// TIA Portal V16 export
// export: Created 2024-12-03T15:41:41.2290419Z, ExportSetting WithDefaults, DisplayName Totally Integrated Automation Portal, DisplayVersion V16 Update 6, DisplayName TIA Portal Version Control Interface, DisplayVersion V16 Update 2, DisplayName TIA Portal Openness, DisplayVersion V16 Update 6, DisplayName TIA Portal Teamcenter Gateway, DisplayVersion V16, DisplayName SINAMICS Startdrive Advanced, DisplayVersion V16 Update 5, DisplayName SINAMICS Startdrive G130, G150, S120, S150, SINAMICS MV, S210, DisplayVersion V16 Update 5, DisplayName SINAMICS Startdrive G110M, G120, G120C, G120D, G120P, G115D, DisplayVersion V16 Update 5, DisplayName STEP 7 Professional, DisplayVersion V16 Update 6, DisplayName STEP 7 Safety, DisplayVersion V16, DisplayName WinCC Advanced / Unified PC, DisplayVersion V16 Update 6
FUNCTION_BLOCK "ConnectionChecker_FB"   // FB13, SCL
{ S7_Optimized_Access := 'TRUE' }
VERSION : 0.1
// stored: AutoNumber true, IsIECCheckEnabled false, IsRetainMemResEnabled false, MemoryReserve 100, SetENOAutomatically false, UDAEnableTagReadback false
   VAR_INPUT
      I_Beat : Word;
      I_Name : String[50];
      I_delay : Time := t#10s;
   END_VAR
   VAR_OUTPUT
      O_alarmActive : Bool;
   END_VAR
   VAR
      prevBeat : Word;
      delay : TON_TIME;
      alarm : Program_Alarm;
   END_VAR
BEGIN
   REGION DETECT ALARM
       #delay(IN := #I_Beat = #prevBeat,
              PT := T#10s);

       #prevBeat := #I_Beat;

   END_REGION

   REGION TRIGGER ALARM

       IF #delay.Q THEN
           #O_alarmActive := 1;
       END_IF;

       IF "Inputs_DB".Reset_System.LE AND #O_alarmActive THEN
           RESET_TIMER(#delay);
           #O_alarmActive := 0;
       END_IF;

       #alarm(SIG:=#O_alarmActive,
              SD_1:=#I_Name);

   END_REGION
END_FUNCTION_BLOCK
